(* CODESYS project magasraktar_visszavag

Project tree, tasks and I/O mapping:
  Device : CODESYS Control for PFC200 SL, 3S - Smart Software Solutions GmbH, version 4.1.0.0
    application Application
      libraries: Standard, 3.5.18.0 (System)
      task MainTask (cyclic, interval t#20ms, priority 1) calls PLC_PRG, PrgTrig
      ANDRAS/
        data type COLOR
        data type EnuAng
        data type ENURENDEZES
        function block FBLERAK [ST]
        data type FBSZIN_VIZS
        function block FINDER [ST]
        function block HETSZEGMENS [ST]
        data type LERAK
        function block RENDEZES [ST]
      function BETWEEN [ST]
      function block FbSzinVizsg [ST]
      global variables GVL
      global variables I
      MAGOCSI/
        function block FBFELVESZ [ST]
        function block FBHIBA [ST]
        function block FBMOZGAS [ST]
        data type FELVESZ_STATE
        data type HIBA_STATE
        data type MOZGAS_STATE
      program PLC_PRG [ST]
      program PrgTrig [ST]
      global variables Q
      data type STATE
      function block VILLOGO4 [ST]
    Pfc200Bus : Wago PFC200 internal bus, 3S - Smart Software Solutions GmbH, version 4.1.0.0
      _750_14xx_1 : 16DI, WAGO Kontakttechnik GmbH u. Co. KG, order no. 750-14xx, version 4.1.0.0
          unmapped channels: %IW10 Digital Inputs 0 - 15
      _750_14xx : 16DI, WAGO Kontakttechnik GmbH u. Co. KG, order no. 750-14xx, version 4.1.0.0
          unmapped channels: %IW5 Digital Inputs 0 - 15
      _750_15xx_1 : 16DO, WAGO Kontakttechnik GmbH u. Co. KG, order no. 750-15xx, version 4.1.0.0
          unmapped channels: %QW10 Digital Outputs 0 - 15
      _750_15xx : 16DO, WAGO Kontakttechnik GmbH u. Co. KG, order no. 750-15xx, version 4.1.0.0
          unmapped channels: %QW5 Digital Outputs 0 - 15
      _75x_459 : 75x-459/0..-000 4AI, 0-10 V, WAGO Kontakttechnik GmbH u. Co. KG, order no. 75x-459(/0..-000), version 4.1.0.0
          unmapped channels: Analog Input Channel 0, Analog Input Channel 1, Analog Input Channel 2, Analog Input Channel 3
      _75x_559 : 75x-559/0..-000 4AO, 0-10 V, WAGO Kontakttechnik GmbH u. Co. KG, order no. 75x-559(/0..-000), version 4.1.0.0
          unmapped channels: Analog Output Channel 0, Analog Output Channel 1, Analog Output Channel 2, Analog Output Channel 3
  function BETWEEN [ST]
  function block VILLOGO4 [ST]
*)

// Device/Application/STATE
{attribute 'qualified_only'}
//{attribute 'strict'}
TYPE STATE :
(
    PRESET := 0,
    BERAKODAS_WAIT := 1,
    KIRAKODAS_WAIT := 2,
    HIBA := 3,
    BERAK_SZIN := 4,
    FELVESZ := 5,
    LERAK := 6
);
END_TYPE

// Device/Application/ANDRAS/COLOR
{attribute 'qualified_only'}
{attribute 'strict'}
TYPE COLOR :
(
	M := 0,
	EZUST := 1,
	FEKETE := 2,
	PIROS := 3
);
END_TYPE

// Device/Application/ANDRAS/EnuAng
{attribute 'qualified_only'}
//{attribute 'strict'}
TYPE EnuAng :
(
	A,
	B,
	C,
	D,
	E,
	F,
	G,
	H
);
END_TYPE

// Device/Application/ANDRAS/ENURENDEZES
{attribute 'qualified_only'}
//{attribute 'strict'}
TYPE ENURENDEZES:
(
	PRESET := 0,
	KERESES := 1,
	MEGFOG := 2,
	LERAKAS := 3,
	HIBA := 4,
	DONE := 5
);
END_TYPE

// Device/Application/ANDRAS/FBSZIN_VIZS
{attribute 'qualified_only'}
//{attribute 'strict'}
TYPE FBSZIN_VIZS:
(
    PRESET := 0,
    KITOL := 1,
    VIZSGAL := 2,
    VISSZA := 3,
    DONE := 4,
	MOVE_SZINV := 5
);
END_TYPE

// Device/Application/ANDRAS/LERAK
{attribute 'qualified_only'}
//{attribute 'strict'}
TYPE LERAK:
(
    PRESET := 0,
    MOVE_LERAK := 1,
    KITOL := 2,
    ELENGED := 3,
    VISSZA_HUZ := 4,
    DONE := 5
	
);
END_TYPE

// Device/Application/MAGOCSI/FELVESZ_STATE
{attribute 'qualified_only'}
//{attribute 'strict'}
TYPE FELVESZ_STATE:
(
    PRESET := 0,
    ODAMEGY := 1,
    KINYUL := 2,
    MEGFOG := 3,
    FELEMEL := 4,
    VISSZAHUZ := 5,
    DONE := 6
);
END_TYPE

// Device/Application/MAGOCSI/HIBA_STATE
{attribute 'qualified_only'}
//{attribute 'strict'}
TYPE HIBA_STATE:
(
    PRESET := 0,
    MEGNYOMVA := 1,
    ELENGEDVE := 2
);
END_TYPE

// Device/Application/MAGOCSI/MOZGAS_STATE
{attribute 'qualified_only'}
//{attribute 'strict'}
TYPE MOZGAS_STATE:
(
    PRESET := 0,
    ANGULARIS_POS := 1,
    AXIALIS_POS := 2,
    ANGULARIS_START := 3,
    AXIALIS_START := 4,
    ANGULARIS_WAIT := 5,
    AXIALIS_WAIT := 6,
    DONE := 7
);
END_TYPE

// Device/Application/GVL
{attribute 'qualified_only'}
VAR_GLOBAL
	MOZGAS_STATE : MOZGAS_STATE;
	CURRENT_ANG : enuAng;
	CURRENT_AXI : INT;
	FELVESZ_STATE : FELVESZ_STATE;
	HIBA_STATE : HIBA_STATE;
   START_R_TRIG : R_TRIG;
   START_F_TRIG : F_TRIG;
   STOP_R_TRIG : R_TRIG;
   STOP_F_TRIG : F_TRIG;
   MODE_R_TRIG : R_TRIG;
   MODE_F_TRIG : F_TRIG;
   PRES_R_TRIG : R_TRIG;
   PRES_F_TRIG : F_TRIG;
   REQ_A_R_TRIG : R_TRIG;
   REQ_A_F_TRIG : F_TRIG;
   REQ_B_R_TRIG : R_TRIG;
   REQ_B_F_TRIG : F_TRIG;
   COL_A_R_TRIG : R_TRIG;
   COL_A_F_TRIG : F_TRIG;
   COL_B_R_TRIG : R_TRIG;
   COL_B_F_TRIG : F_TRIG;
   RAD_OFF_R_TRIG : R_TRIG;
   RAD_OFF_F_TRIG : F_TRIG;
   RAD_ON0_R_TRIG : R_TRIG;
   RAD_ON0_F_TRIG : F_TRIG;
   AXI_RDY_R_TRIG : R_TRIG;
   AXI_RDY_F_TRIG : F_TRIG;
   ANG_RDY_R_TRIG : R_TRIG;
   ANG_RDY_F_TRIG : F_TRIG;
   
   COLOR : COLOR;
   state :state;
   lerak : lerak;
   FBSZIN_VIZS : FBSZIN_VIZS;
   	ANG : enuAng;
	AXI : INT;
	RAKTAR : ARRAY [1..3, 0..5] OF BOOL;
END_VAR

// Device/Application/I
{attribute 'qualified_only'}
VAR_GLOBAL
   START AT %IX20.0 : BOOL;
   STOP_NC AT %IX20.1 : BOOL;
   STOP : BOOL;
   MODE AT %IX20.2 : BOOL;
   PRES AT %IX20.3 : BOOL;
   REQ_A AT %IX20.4 : BOOL;
   REQ_B AT %IX20.5 : BOOL;
   COL_A AT %IX20.6 : BOOL;
   COL_B AT %IX20.7 : BOOL;
   RAD_OFF AT %IX21.0 : BOOL;
   RAD_ON AT %IX21.1 : BOOL;
   AXI_RDY AT %IX21.2 : BOOL;
   ANG_RDY AT %IX21.3 : BOOL;




END_VAR

// Device/Application/Q
{attribute 'qualified_only'}
VAR_GLOBAL
END_VAR

// Device/Application/PLC_PRG
PROGRAM PLC_PRG
VAR
	
    DONE : BOOL;
    FBFELVESZEM : FBFELVESZ;
    FBLERAKAS : FBLERAK;
    FBPRESET : FBMOZGAS;
    FBSZIN : FBSZINVIZSG;
    HIBA : FBHIBA;
    TELE : BOOL;
    VALID_SZIN : BOOL;
	INDEX : INT;
	stop_mem : BOOL;
	
	FINDEEEE : FINDER;
	
	
END_VAR

IF i.STOP THEN
	stop_mem := TRUE;
END_IF


CASE GVL.STATE OF

    STATE.PRESET:
	q.GRIP := FALSE;
	q.RAD := false;
	stop_mem := false;
	FBPRESET(EN:= (GVL.STATE = STATE.PRESET) , ang := ENUANG.H , axi := 7 );
	
    IF FBPRESET.DONE AND NOT I.MODE THEN
        GVL.STATE := STATE.BERAKODAS_WAIT;
    ELSIF FBPRESET.DONE AND I.MODE THEN
        GVL.STATE := STATE.KIRAKODAS_WAIT;
    END_IF


    STATE.BERAKODAS_WAIT:
	
    IF I.MODE THEN
        GVL.STATE := STATE.KIRAKODAS_WAIT;
    ELSIF I.START THEN
        GVL.STATE := STATE.BERAK_SZIN;
    END_IF

    STATE.KIRAKODAS_WAIT:
    //KERES RÖGZITÉS
	
    IF NOT I.MODE THEN
        GVL.STATE := STATE.BERAKODAS_WAIT;
    END_IF
	
	 

    STATE.HIBA:
	
    IF HIBA.ACK THEN
        GVL.STATE := STATE.PRESET;
    END_IF

   STATE.BERAK_SZIN:
   IF FBSZIN.DONE AND NOT (GVL.COLOR = COLOR.M)  THEN
	   VALID_SZIN := TRUE;
	ELSE
		 VALID_SZIN := FALSE;
   END_IF
   
   
   	IF FBSZIN.DONE AND VALID_SZIN THEN

	FOR INDEX := 5 TO 0 BY -1 DO
		IF NOT GVL.RAKTAR[GVL.COLOR,INDEX] THEN
			TELE := FALSE;
			EXIT;
		ELSE
			TELE := TRUE;
		END_IF
	END_FOR   
	END_IF
  
    IF FBSZIN.DONE AND VALID_SZIN AND NOT TELE THEN
		GVL.ANG := ENUANG.G;
		GVL.AXI := 7;
        GVL.STATE := STATE.FELVESZ;
    ELSIF FBSZIN.DONE AND NOT VALID_SZIN THEN
        GVL.STATE := STATE.PRESET;
    ELSIF FBSZIN.DONE AND VALID_SZIN AND TELE THEN
        GVL.STATE := STATE.HIBA;
    END_IF

    STATE.FELVESZ:

    IF FBFELVESZEM.DONE THEN
		GVL.ANG := INDEX;
		CASE GVL.COLOR OF
			COLOR.PIROS:
			GVL.AXI := 1;
			COLOR.EZUST:
			GVL.AXI := 3;
			COLOR.FEKETE:
			GVL.AXI := 6;
		END_CASE
        GVL.STATE := STATE.LERAK;
    END_IF

    STATE.LERAK:

    IF FBLERAKAS.DONE AND NOT stop_mem THEN
		GVL.RAKTAR[GVL.COLOR, INDEX] := TRUE;
        GVL.STATE := STATE.BERAK_SZIN;
    END_IF
	
	IF stop_mem and FBLERAKAS.DONE THEN
		GVL.RAKTAR[GVL.COLOR, INDEX] := TRUE;
	GVL.STATE := STATE.PRESET;
	END_IF

END_CASE


FBFELVESZEM(EN:= (GVL.STATE = STATE.FELVESZ) , ang := gvl.ANG , axi := gvl.AXI);
HIBA(EN:= (GVL.STATE = STATE.HIBA));
FBLERAKAS(EN:= (GVL.STATE = STATE.LERAK) , ang := gvl.ANG , axi := gvl.AXI );

FBSZIN(EN:= (GVL.STATE = STATE.BERAK_SZIN) );

q.ERROR := gvl.state = state.HIBA;

FINDEEEE(EN := TRUE , SZIN := COLOR.FEKETE );

END_PROGRAM

// Device/Application/MAGOCSI/FBFELVESZ
FUNCTION_BLOCK FBFELVESZ
VAR_INPUT
	EN : BOOL;
	ANG : INT;
	AXI : INT;
END_VAR
VAR_OUTPUT
    DONE  : BOOL;
END_VAR
VAR
	NEW_AXI : INT;
    MOZOG : FBMOZGAS;
    TRANS_MEGFOG_FELEMEL_T : TON;
END_VAR

IF NOT EN THEN
	GVL.FELVESZ_STATE := FELVESZ_STATE.PRESET;
	DONE := FALSE;
	RETURN;
END_IF

TRANS_MEGFOG_FELEMEL_T(PT:= T#1S, IN:= (GVL.FELVESZ_STATE = FELVESZ_STATE.MEGFOG));
MOZOG(ANG := ANG, AXI := NEW_AXI, EN:= (GVL.FELVESZ_STATE = FELVESZ_STATE.FELEMEL) OR (GVL.FELVESZ_STATE = FELVESZ_STATE.ODAMEGY));

CASE GVL.FELVESZ_STATE OF

    FELVESZ_STATE.PRESET:

    IF TRUE THEN
        GVL.FELVESZ_STATE := FELVESZ_STATE.ODAMEGY;
    END_IF


    FELVESZ_STATE.ODAMEGY:

    IF MOZOG.DONE THEN
		NEW_AXI := NEW_AXI - 1;
        GVL.FELVESZ_STATE := FELVESZ_STATE.KINYUL;
    END_IF


    FELVESZ_STATE.KINYUL:

    IF I.RAD_ON THEN
        GVL.FELVESZ_STATE := FELVESZ_STATE.MEGFOG;
    END_IF

    FELVESZ_STATE.MEGFOG:
    Q.GRIP := TRUE;

    IF TRANS_MEGFOG_FELEMEL_T.Q THEN
        GVL.FELVESZ_STATE := FELVESZ_STATE.FELEMEL;
    END_IF


    FELVESZ_STATE.FELEMEL:

    IF MOZOG.DONE THEN
        GVL.FELVESZ_STATE := FELVESZ_STATE.VISSZAHUZ;
    END_IF


    FELVESZ_STATE.VISSZAHUZ:

    IF I.RAD_OFF THEN
        GVL.FELVESZ_STATE := FELVESZ_STATE.DONE;
    END_IF


END_CASE

DONE := (GVL.FELVESZ_STATE = FELVESZ_STATE.DONE);
Q.RAD := (GVL.FELVESZ_STATE = FELVESZ_STATE.FELEMEL) OR (GVL.FELVESZ_STATE = FELVESZ_STATE.KINYUL) OR (GVL.FELVESZ_STATE = FELVESZ_STATE.MEGFOG);

END_FUNCTION_BLOCK

// Device/Application/MAGOCSI/FBMOZGAS
FUNCTION_BLOCK FBMOZGAS
VAR_INPUT
    ANG : enuang;
	AXI : INT;
	EN : BOOL;
END_VAR
VAR_OUTPUT
    DONE  : BOOL;
END_VAR
VAR
    TRANS_ANGULARIS_POS_ANGULARIS_START_T : TON;
    TRANS_ANGULARIS_START_ANGULARIS_WAIT_T : TON;
    TRANS_AXIALIS_POS_AXIALIS_START_T : TON;
    TRANS_AXIALIS_START_AXIALIS_WAIT_T : TON;
END_VAR

IF NOT EN THEN
	GVL.MOZGAS_STATE := MOZGAS_STATE.PRESET;
	DONE := FALSE;
	RETURN;
END_IF

TRANS_AXIALIS_START_AXIALIS_WAIT_T(PT:= T#200MS, IN:= (GVL.MOZGAS_STATE = MOZGAS_STATE.AXIALIS_START));
TRANS_ANGULARIS_START_ANGULARIS_WAIT_T(PT:= T#200MS, IN:= (GVL.MOZGAS_STATE = MOZGAS_STATE.ANGULARIS_START));
TRANS_AXIALIS_POS_AXIALIS_START_T(PT:= T#50MS, IN:= (GVL.MOZGAS_STATE = MOZGAS_STATE.AXIALIS_POS));
TRANS_ANGULARIS_POS_ANGULARIS_START_T(PT:= T#50MS, IN:= (GVL.MOZGAS_STATE = MOZGAS_STATE.ANGULARIS_POS));

CASE GVL.MOZGAS_STATE OF

    MOZGAS_STATE.PRESET:

    IF NOT (ANG = GVL.CURRENT_ANG) THEN
        GVL.MOZGAS_STATE := MOZGAS_STATE.ANGULARIS_POS;
    ELSIF ANG = GVL.CURRENT_ANG THEN
        GVL.MOZGAS_STATE := MOZGAS_STATE.AXIALIS_POS;
    END_IF

    MOZGAS_STATE.ANGULARIS_POS:
    Q.POS_A := ANG.0;
    Q.POS_B := ANG.1;
    Q.POS_C := ANG.2;

    IF TRANS_ANGULARIS_POS_ANGULARIS_START_T.Q THEN
        GVL.MOZGAS_STATE := MOZGAS_STATE.ANGULARIS_START;
    END_IF

    MOZGAS_STATE.AXIALIS_POS:
    Q.POS_A := AXI.0;
    Q.POS_B := AXI.1;
    Q.POS_C := AXI.2;

    IF TRANS_AXIALIS_POS_AXIALIS_START_T.Q THEN
        GVL.MOZGAS_STATE := MOZGAS_STATE.AXIALIS_START;
    END_IF


    MOZGAS_STATE.ANGULARIS_START:

    IF TRANS_ANGULARIS_START_ANGULARIS_WAIT_T.Q THEN
        GVL.MOZGAS_STATE := MOZGAS_STATE.ANGULARIS_WAIT;
    END_IF


    MOZGAS_STATE.AXIALIS_START:

    IF TRANS_AXIALIS_START_AXIALIS_WAIT_T.Q THEN
        GVL.MOZGAS_STATE := MOZGAS_STATE.AXIALIS_WAIT;
    END_IF


    MOZGAS_STATE.ANGULARIS_WAIT:

    IF I.ANG_RDY THEN
        GVL.MOZGAS_STATE := MOZGAS_STATE.AXIALIS_POS;
    END_IF


    MOZGAS_STATE.AXIALIS_WAIT:

    IF I.AXI_RDY THEN
		gvl.CURRENT_ANG := ang; 
		gvl.CURRENT_AXI := axi;
        GVL.MOZGAS_STATE := MOZGAS_STATE.DONE;
    END_IF


END_CASE

DONE := (GVL.MOZGAS_STATE = MOZGAS_STATE.DONE);
Q.ANG_ST := (GVL.MOZGAS_STATE = MOZGAS_STATE.ANGULARIS_START);
Q.AXI_ST := (GVL.MOZGAS_STATE = MOZGAS_STATE.AXIALIS_START);

END_FUNCTION_BLOCK

// Device/Application/ANDRAS/FBLERAK
FUNCTION_BLOCK FBLERAK
VAR_INPUT
	
	EN : BOOL;
	ANG : EnuAng;
    AXI : INT;
	
END_VAR
VAR_OUTPUT
END_VAR
VAR
	TRANS_ELENGED_VISSZA_HUZ_T : TON;
	LERAK : LERAK;
	FBMOZGATAS : FBMOZGAS;
END_VAR



IF NOT EN THEN
	LERAK := LERAK.PRESET
	RETURN;
END_IF

RANS_ELENGED_VISSZA_HUZ_T(PT:= T#1S, IN:= (LERAK = LERAK.ELENGED));
FBMOZGATAS(EN := (LERAK = LERAK.MOVE_LERAK ) ,ANG := ANG, AXI := AXI);

CASE LERAK OF

    LERAK.PRESET:

    IF EN THEN
        GVL.LERAK := LERAK.MOVE_LERAK;
    END_IF

    LERAK.MOVE_LERAK:

    IF FBMOZGATAS.DONE THEN
        GVL.LERAK := LERAK.KITOL;
    END_IF

    LERAK.KITOL:

    IF I.RAD_ON THEN
        GVL.LERAK := LERAK.ELENGED;
    END_IF

    LERAK.ELENGED:
    Q.GRIP := FALSE;

    IF TRANS_ELENGED_VISSZA_HUZ_T.Q THEN
        GVL.LERAK := LERAK.VISSZA_HUZ;
    END_IF


    LERAK.VISSZA_HUZ:

    IF I.RAD_OFF THEN
        GVL.LERAK := LERAK.DONE;
    END_IF
	
	
	

END_CASE

Q.RAD := (GVL.LERAK = LERAK.KITOL);
DONE := LERAK = LERAK.DONE;

END_FUNCTION_BLOCK

// Device/Application/FbSzinVizsg
FUNCTION_BLOCK FbSzinVizsg
VAR_INPUT
	EN:BOOL;
END_VAR
VAR_OUTPUT
	DONE:BOOL;
END_VAR
VAR
	    TRANS_VIZSGAL_VISSZA_T : TON;
		FBSZIN_VIZS : FBSZIN_VIZS;
END_VAR

TRANS_VIZSGAL_VISSZA_T(PT:= T#1S, IN:= (FBSZIN_VIZS = FBSZIN_VIZS.VIZSGAL));

CASE FBSZIN_VIZS OF

    FBSZIN_VIZS.PRESET:

    IF EN THEN
        GVL.FBSZIN_VIZS := FBSZIN_VIZS.KITOL;
    END_IF


    FBSZIN_VIZS.KITOL:

    IF I.RAD_ON THEN
        GVL.FBSZIN_VIZS := FBSZIN_VIZS.VIZSGAL;
    END_IF

   FBSZIN_VIZS.VIZSGAL:
   
    GVL.COLOR.0 := I.COL_A;
    GVL.COLOR.1 := I.COL_B;

    IF TRANS_VIZSGAL_VISSZA_T.Q THEN
        GVL.FBSZIN_VIZS := FBSZIN_VIZS.VISSZA;
    END_IF


    FBSZIN_VIZS.VISSZA:

    IF I.RAD_OFF THEN
        GVL.FBSZIN_VIZS := FBSZIN_VIZS.DONE;
    END_IF


END_CASE

DONE := (FBSZIN_VIZS = FBSZIN_VIZS.DONE);
Q.RAD := (FBSZIN_VIZS = FBSZIN_VIZS.KITOL) OR (FBSZIN_VIZS = FBSZIN_VIZS.VIZSGAL);

END_FUNCTION_BLOCK

// Device/Application/MAGOCSI/FBHIBA
FUNCTION_BLOCK FBHIBA
VAR_INPUT
	EN : BOOL;
END_VAR
VAR_OUTPUT
	ACK : BOOL ; 
END_VAR
VAR
END_VAR

IF NOT EN THEN
	GVL.HIBA_STATE := HIBA_STATE.PRESET;
	ACK := FALSE;
	RETURN;
END_IF

CASE GVL.HIBA_STATE OF

    HIBA_STATE.PRESET:

    IF GVL.STOP_R_TRIG.Q THEN
        GVL.HIBA_STATE := HIBA_STATE.MEGNYOMVA;
    END_IF


    HIBA_STATE.MEGNYOMVA:

    IF GVL.STOP_F_TRIG.Q THEN
        GVL.HIBA_STATE := HIBA_STATE.ELENGEDVE;
    END_IF


END_CASE

ACK := (GVL.HIBA_STATE = HIBA_STATE.ELENGEDVE);

END_FUNCTION_BLOCK

// Device/Application/ANDRAS/FINDER
FUNCTION_BLOCK FINDER
VAR_INPUT
	SZIN : COLOR;
	EN : BOOL;
END_VAR
VAR_OUTPUT
	ANG : ENUANG;
	ELSO_URES : ENUANG;
	ELSO_FELVENNI : ENUANG;
	DONE : BOOL;
	RENDEZVE : BOOL;
END_VAR
VAR
	INDEX : INT;
	ELSO_URES_MEM : INT := -1;
END_VAR

IF NOT  EN THEN
	DONE := FALSE;
	RENDEZVE := FALSE;
	ELSO_URES_MEM := -1;
	RETURN ;
END_IF


FOR INDEX := 5 TO -1 BY -1 DO
	IF 	INDEX = -1 THEN
		RENDEZVE := TRUE;
		RETURN;
	END_IF

	IF (GVL.RAKTAR[SZIN,INDEX] = FALSE) AND (ELSO_URES_MEM = -1) THEN
		ELSO_URES_MEM := INDEX;
	END_IF
	
	IF ELSO_URES_MEM <> 0 AND GVL.RAKTAR[SZIN,INDEX] THEN
		ELSO_FELVENNI := INDEX;
		ELSO_URES := ELSO_URES_MEM;
		RETURN;
	END_IF
	
END_FOR

RETURN;

END_FUNCTION_BLOCK

// Device/Application/PrgTrig
PROGRAM PrgTrig
VAR
END_VAR

GVL.START_R_TRIG(CLK:= I.START);
GVL.START_F_TRIG(CLK:= I.START);
I.STOP := NOT I.STOP_NC;
GVL.STOP_R_TRIG(CLK:= I.STOP);
GVL.STOP_F_TRIG(CLK:= I.STOP);
GVL.MODE_R_TRIG(CLK:= I.MODE);
GVL.MODE_F_TRIG(CLK:= I.MODE);
GVL.PRES_R_TRIG(CLK:= I.PRES);
GVL.PRES_F_TRIG(CLK:= I.PRES);
GVL.REQ_A_R_TRIG(CLK:= I.REQ_A);
GVL.REQ_A_F_TRIG(CLK:= I.REQ_A);
GVL.REQ_B_R_TRIG(CLK:= I.REQ_B);
GVL.REQ_B_F_TRIG(CLK:= I.REQ_B);
GVL.COL_A_R_TRIG(CLK:= I.COL_A);
GVL.COL_A_F_TRIG(CLK:= I.COL_A);
GVL.COL_B_R_TRIG(CLK:= I.COL_B);
GVL.COL_B_F_TRIG(CLK:= I.COL_B);
GVL.RAD_OFF_R_TRIG(CLK:= I.RAD_OFF);
GVL.RAD_OFF_F_TRIG(CLK:= I.RAD_OFF);
GVL.RAD_ON0_R_TRIG(CLK:= I.RAD_ON0);
GVL.RAD_ON0_F_TRIG(CLK:= I.RAD_ON0);
GVL.AXI_RDY_R_TRIG(CLK:= I.AXI_RDY);
GVL.AXI_RDY_F_TRIG(CLK:= I.AXI_RDY);
GVL.ANG_RDY_R_TRIG(CLK:= I.ANG_RDY);
GVL.ANG_RDY_F_TRIG(CLK:= I.ANG_RDY);

END_PROGRAM

// BETWEEN
FUNCTION BETWEEN : BOOL
VAR_INPUT
	STATE : INT;
	LOW : INT;
	HIGH : INT;
END_VAR
VAR_OUTPUT
END_VAR
VAR
	EN_TRIG : F_TRIG;
END_VAR

IF STATE >= LOW AND STATE <= HIGH THEN
	BETWEEN := TRUE;
ELSE 
	BETWEEN := FALSE;
END_IF

END_FUNCTION

// Device/Application/BETWEEN
FUNCTION BETWEEN : BOOL
VAR_INPUT
	STATE : INT;
	LOW : INT;
	HIGH : INT;
END_VAR
VAR_OUTPUT
END_VAR
VAR
	EN_TRIG : F_TRIG;
END_VAR

IF STATE >= LOW AND STATE <= HIGH THEN
	BETWEEN := TRUE;
ELSE 
	BETWEEN := FALSE;
END_IF

END_FUNCTION

// VILLOGO4
FUNCTION_BLOCK VILLOGO4
VAR_INPUT
	T1: TIME;
	T2: TIME;
	T3: TIME;
	T4: TIME;
END_VAR
VAR_IN_OUT
	Q1: BOOL;
	Q2: BOOL;
	Q3: BOOL;
	Q4: BOOL;
END_VAR
VAR
	T1_TON: TON;
	T2_TON: TON;
	T3_TON: TON;
	T4_TON: TON;
END_VAR
VAR_INPUT
	EN: BOOL := FALSE;
END_VAR
VAR
	EN_F_TRIG: F_TRIG;
	EN_R_TRIG: R_TRIG;
	STATE: INT := 0;
	PREV_STATE: INT := 0;
END_VAR

EN_F_TRIG(CLK := EN);
EN_R_TRIG(CLK := EN);

IF EN_F_TRIG.Q THEN
	Q1 := FALSE;
	Q2 := FALSE;
	Q3 := FALSE;
	Q4 := FALSE;
	T1_TON.PT := T1_TON.ET;
	T2_TON.PT := T2_TON.ET;
	T3_TON.PT := T3_TON.ET;
	T4_TON.PT := T4_TON.ET;
	STATE := 0;
ELSIF EN_R_TRIG.Q THEN
		Q1 := TRUE;
END_IF

IF NOT EN THEN
	RETURN;
END_IF

T1_TON(IN:= EN_R_TRIG.Q OR (STATE = 0), PT:= T1);
T2_TON(IN:= STATE = 1, PT:= T2);
T3_TON(IN:= STATE = 2, PT:= T3);
T4_TON(IN:= STATE = 3, PT:= T4);

IF T1_TON.Q THEN
	Q1 := FALSE;
	Q2 := TRUE;
END_IF
IF T2_TON.Q THEN
	Q2 := FALSE;
	Q3 := TRUE;
END_IF
IF T3_TON.Q THEN
	Q3 := FALSE;
	Q4 := TRUE;
END_IF
IF T4_TON.Q THEN
	Q4 := FALSE;
	Q1 := TRUE;
END_IF

IF T1_TON.Q OR T2_TON.Q OR T3_TON.Q OR T4_TON.Q THEN
	STATE := STATE + 1;
END_IF

IF STATE > 3 THEN
	STATE := 0;
END_IF

END_FUNCTION_BLOCK

// Device/Application/VILLOGO4
FUNCTION_BLOCK VILLOGO4
VAR_INPUT
	T1: TIME;
	T2: TIME;
	T3: TIME;
	T4: TIME;
END_VAR
VAR_IN_OUT
	Q1: BOOL;
	Q2: BOOL;
	Q3: BOOL;
	Q4: BOOL;
END_VAR
VAR
	T1_TON: TON;
	T2_TON: TON;
	T3_TON: TON;
	T4_TON: TON;
END_VAR
VAR_INPUT
	EN: BOOL := FALSE;
END_VAR
VAR
	EN_F_TRIG: F_TRIG;
	EN_R_TRIG: R_TRIG;
	STATE: INT := 0;
	PREV_STATE: INT := 0;
END_VAR

EN_F_TRIG(CLK := EN);
EN_R_TRIG(CLK := EN);

IF EN_F_TRIG.Q THEN
	Q1 := FALSE;
	Q2 := FALSE;
	Q3 := FALSE;
	Q4 := FALSE;
	T1_TON.PT := T1_TON.ET;
	T2_TON.PT := T2_TON.ET;
	T3_TON.PT := T3_TON.ET;
	T4_TON.PT := T4_TON.ET;
	STATE := 0;
ELSIF EN_R_TRIG.Q THEN
		Q1 := TRUE;
END_IF

IF NOT EN THEN
	RETURN;
END_IF

T1_TON(IN:= EN_R_TRIG.Q OR (STATE = 0), PT:= T1);
T2_TON(IN:= STATE = 1, PT:= T2);
T3_TON(IN:= STATE = 2, PT:= T3);
T4_TON(IN:= STATE = 3, PT:= T4);

IF T1_TON.Q THEN
	Q1 := FALSE;
	Q2 := TRUE;
END_IF
IF T2_TON.Q THEN
	Q2 := FALSE;
	Q3 := TRUE;
END_IF
IF T3_TON.Q THEN
	Q3 := FALSE;
	Q4 := TRUE;
END_IF
IF T4_TON.Q THEN
	Q4 := FALSE;
	Q1 := TRUE;
END_IF

IF T1_TON.Q OR T2_TON.Q OR T3_TON.Q OR T4_TON.Q THEN
	STATE := STATE + 1;
END_IF

IF STATE > 3 THEN
	STATE := 0;
END_IF

END_FUNCTION_BLOCK

// Device/Application/ANDRAS/HETSZEGMENS
FUNCTION_BLOCK HETSZEGMENS
VAR_INPUT
	en : BOOL;
	color_mode : BOOL;
	index_mode : BOOL;
	index : INT;
	szin : color;
END_VAR
VAR_OUTPUT
END_VAR
VAR
END_VAR

IF NOT en THEN
	q.SS_A := FALSE;
	q.SS_B := FALSE;
	q.SS_C := FALSE;
	RETURN;
END_IF


IF color_mode THEN
	CASE szin OF
		color.PIROS:
			q.SS_A := TRUE;
			q.SS_B := FALSE;
			q.SS_C := TRUE;
		color.EZUST:
			q.SS_A := FALSE;
			q.SS_B := TRUE;
			q.SS_C := TRUE;
		color.FEKETE:
			q.SS_A := TRUE;
			q.SS_B := TRUE;
			q.SS_C := TRUE;
	END_CASE
	RETURN;
	
END_IF

IF index_mode THEN
	q.SS_A := index.0;
	q.SS_B := index.1;
	q.SS_C := index.2;
	RETURN;
END_IF

END_FUNCTION_BLOCK

// Device/Application/ANDRAS/RENDEZES
FUNCTION_BLOCK RENDEZES
VAR_INPUT
END_VAR
VAR_OUTPUT
	DONE : BOOL;
END_VAR
VAR
	FINDE : FINDER;
	BAJVAN : BOOL;
	EN : BOOL;
	FELVETEL : FBFELVESZ;;
	LERAKODAS : FBLERAK;
	RENDEZES : ENURENDEZES;
	FASZA :BOOL;
	SZIN : COLOR := COLOR.EZUST;
	
	AXI : INT;
	ANG : ENUANG;
END_VAR

IF NOT EN THEN
	RENDEZES := ENURENDEZES.PRESET;
	FASZA := FALSE;
	DONE := FALSE;
	RETURN;
END_IF

IF BAJVAN THEN
	RENDEZES := ENURENDEZES.HIBA;
END_IF

FELVETEL(EN:= (RENDEZES = ENURENDEZES.MEGFOG) ,AXI := AXI , ANG := ANG);
LERAKODAS(EN:= (RENDEZES = ENURENDEZES.LERAKAS) ,AXI := AXI , ANG := ANG);
FINDE(EN:= (RENDEZES = ENURENDEZES.KERESES) , SZIN := SZIN);

CASE RENDEZES OF

	ENURENDEZES.PRESET:

	IF EN THEN
		RENDEZES := ENURENDEZES.KERESES;
	END_IF

	ENURENDEZES.KERESES:
	
	//HA BERENDEZET COLOR VÁLTÁS  ÉS MÉGEGYSZER FINDER
	//HA MINDEN FQASZA DONE
	

	IF FINDE.DONE AND NOT FINDER.RENDEZVE THEN
		AXI := SZIN;
		ANG := FINDER.ELSO_FELVENNI;
		RENDEZES := ENURENDEZES.MEGFOG;
	ELSIF FINDER.RENDEZVE AND SZIN = COLOR.PIROS THEN
		RENDEZES := ENURENDEZES.DONE;
	ELSIF (NOT (SZIN = COLOR.PIROS) ) AND FINDER.RENDEZVE THEN
		RENDEZES := ENURENDEZES.PRESET;
	END_IF

	ENURENDEZES.MEGFOG:
	//ANG AXI IRÁSA

	IF FELVETEL.DONE THEN
		AXI := SZIN;
		ANG := FINDER.ELSO_URES;
		RENDEZES := ENURENDEZES.LERAKAS;
	END_IF

	ENURENDEZES.LERAKAS:
	//ANG AXI IRÁSA

	IF LERAKODAS.DONE THEN
		RENDEZES := ENURENDEZES.KERESES;
	END_IF
	
	ENURENDEZES.DONE:
	DONE := TRUE;




END_CASE

END_FUNCTION_BLOCK
